{attribute 'TcGenerated'}
{attribute 'no-analysis'}
{attribute 'linkalways'}
// This function has been automatically generated from the project information.
VAR_GLOBAL CONSTANT
    {attribute 'const_non_replaced'}
    stLibVersion_LibraryVision : ST_LibVersion :=
    (
        iMajor      := 0
        , iMinor    := 9
        , iBuild    := 9
        , iRevision := 9
        , nFlags    := 0
        , sVersion  := '0.9.9.9'
    );
END_VAR

(* stored: Version 1.1.0.1, ProductVersion 3.1.4024.12
   GVL Global_Version: Id {87be6246-8890-4d67-a158-b36bf2a2b9bf} *)
